(*
SPDX-FileCopyrightText: Â© 2026 Oleksandr Tiutyk <trofimich@gmail.com>
SPDX-License-Identifier: MIT
License: https://opensource.org/license/mit
*)

(*!
<summary>Read-only contract for an analog output automation component.</summary>
<description>
Provides access to engineering output value, assigned converter and raw representation.
</description>
*)

INTERFACE IReadOnlyAnalogOutput EXTENDS TOF_Automation.IOutputLeafAutomationComponent

(*!
<summary>Gets the assigned analog value converter.</summary>
*)
{attribute 'monitoring' := 'call'}
PROPERTY Converter : IAnalogValueConverter
GET
END_GET
END_PROPERTY

(*!
<summary>Gets current raw hardware DAC value cast to LREAL.</summary>
*)
{attribute 'monitoring' := 'call'}
PROPERTY RawValue : LREAL
GET
END_GET
END_PROPERTY

(*!
<summary>Gets the raw analog data representation type.</summary>
*)
{attribute 'monitoring' := 'call'}
PROPERTY RawValueType : RAW_ANALOG_VALUE_TYPE
GET
END_GET
END_PROPERTY

(*!
<summary>Gets current scaled engineering unit output value.</summary>
*)
{attribute 'monitoring' := 'call'}
PROPERTY Value : LREAL
GET
END_GET
END_PROPERTY

END_INTERFACE

(* stored: Version 1.1.0.1
   Itf IReadOnlyAnalogOutput: Id {488a2803-10f4-425a-a5b9-a9ffcf76a2fb}
   Property Converter: Id {7725b43b-8616-4073-9849-d813b6c8da57}
   Get Get: Id {6680ded0-c31d-48e2-a8c4-0b92706159b2}
   Property RawValue: Id {4499d025-563c-4f19-a5dc-101ca2fbbd4d}
   Get Get: Id {2a33335e-ee4f-4963-ae0a-18cad69d38bc}
   Property RawValueType: Id {5436adff-0956-4433-b426-ad5851a54c78}
   Get Get: Id {144c3cce-16c6-445e-8609-6d53d1e16f0e}
   Property Value: Id {cc66aada-ccd0-4b51-9659-0112c159ff08}
   Get Get: Id {d9506307-77fb-4089-82eb-38101583c337} *)
